(*			
	RAFALOS
	Rafał Osajda		19.09.2025		TC 4024.66
	
*)
FUNCTION_BLOCK FB_BaseFlag IMPLEMENTS ITF_BaseFlag
VAR
	bState				: BOOL;
END_VAR

METHOD PUBLIC GetFlag : BOOL
VAR_INPUT
END_VAR
GetFlag			:= THIS^.bState;
END_METHOD

METHOD PUBLIC SetFlag
VAR_INPUT
	bState				: BOOL;
END_VAR
THIS^.bState			:= bState;
END_METHOD

END_FUNCTION_BLOCK

(* stored: Version 1.1.0.1
   POU FB_BaseFlag: Id {4cccc323-b44e-0e45-096d-9e86741e033e}, SpecialFunc None
   Method GetFlag: Id {7e86e6a8-5c6a-0c08-063a-dbd6b6149b83}
   Method SetFlag: Id {37efbdda-7095-09eb-2668-2e143dcbc25c} *)
